// TIA Portal V19 export
FUNCTION "System_CALL" : Void   // FC9, LAD
TITLE = SYSTEM CALL
// stored: SetENOAutomatically false
BEGIN

REGION Network 1: System Call
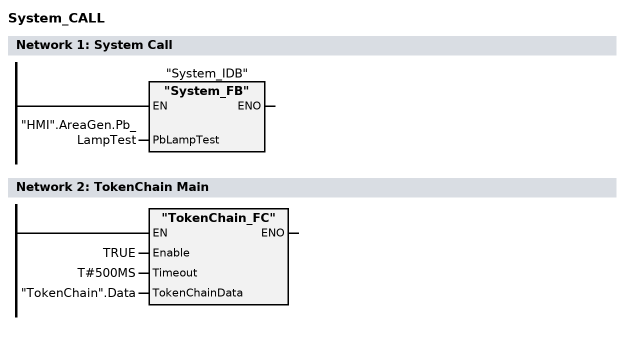
   RUNG wire#powerrail
      "System_IDB"(PbLampTest := "HMI".AreaGen.Pb_LampTest)
   END_RUNG
   // the same network as SCL:
   "System_IDB"(PbLampTest := "HMI".AreaGen.Pb_LampTest);   // "System_FB"
END_REGION

REGION Network 2: TokenChain Main
   RUNG wire#powerrail
      "TokenChain_FC"(Enable := TRUE, Timeout := T#500MS, TokenChainData := "TokenChain".Data)
   END_RUNG
   // the same network as SCL:
   "TokenChain_FC"(Enable := TRUE, Timeout := T#500MS, TokenChainData := "TokenChain".Data);
END_REGION
END_FUNCTION
